ABB RAPID module: Module1.mod

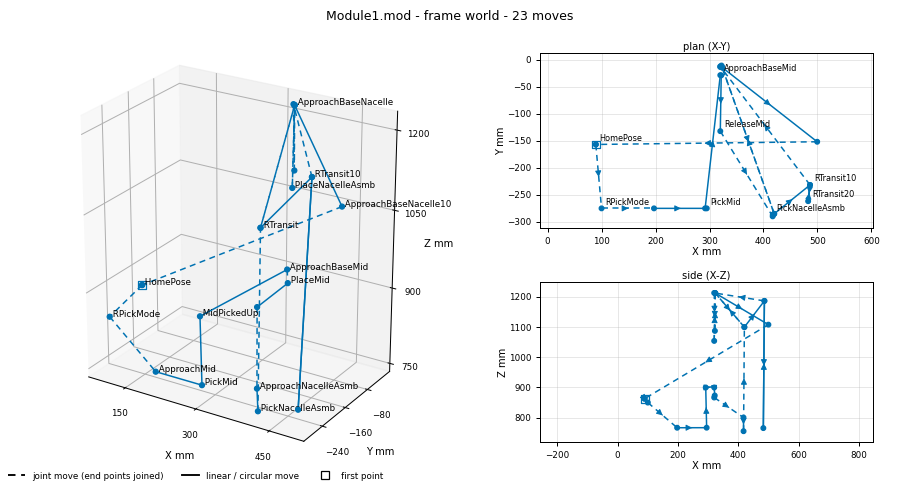
[picture p0: tool path of Module1.mod in frame world, 23 of 23 moves have a stored position in this frame; points joined in program order, loops and branches not executed]
MODULE Module1
    CONST robtarget HomePose:=[[89.387946422,-156.622117956,147.913470217],[0.066010726,-0.842420918,-0.111214912,-0.523068661],[0,0,0,4],[-101.964427132,9E+09,9E+09,9E+09,9E+09,9E+09]];
    CONST robtarget RPickMode:=[[100,-275,135],[0.489762134,0.473830049,0.544432409,0.489092516],[0,0,-1,4],[-101.964427132,9E+09,9E+09,9E+09,9E+09,9E+09]];
    CONST robtarget ApproachMid:=[[-122.697727862,-0.008118871,49.551256125],[0.499992891,0.499992406,0.500008511,0.50000619],[0,0,-1,4],[-101.964431802,9E+09,9E+09,9E+09,9E+09,9E+09]];
    CONST robtarget PickMid:=[[-24.998727784,-0.00024572,49.697076732],[0.499992891,0.499992406,0.500008511,0.50000619],[0,0,-1,4],[-101.964431802,9E+09,9E+09,9E+09,9E+09,9E+09]];
    CONST robtarget MidPickedUp:=[[-27.998642636,0.000176123,182.899085274],[0.499992714,0.499992387,0.500008355,0.500006542],[1,0,-1,4],[-101.964431802,9E+09,9E+09,9E+09,9E+09,9E+09]];
    CONST robtarget ApproachBaseMid:=[[-28.27,0.00,185.00],[0.499997,0.499992,0.500001,0.50001],[1,-1,0,4],[-101.957,9E+09,9E+09,9E+09,9E+09,9E+09]];
    CONST robtarget PlaceMid:=[[-28.61,-1.73,158.37],[0.483819,0.495256,0.51307,0.507346],[1,-1,0,4],[-104.271,9E+09,9E+09,9E+09,9E+09,9E+09]];
    CONST robtarget ReleaseMid:=[[-131.99,0.00,151.74],[0.499992,0.499992,0.500006,0.500009],[1,-1,0,4],[-101.961,9E+09,9E+09,9E+09,9E+09,9E+09]];
    CONST robtarget ApproachNacelleAsmb:=[[15.11,-2.84,84.21],[0.000268004,0.030298,-0.999539,-0.00191911],[1,-2,1,4],[-101.993,9E+09,9E+09,9E+09,9E+09,9E+09]];
    CONST robtarget PickNacelleAsmb:=[[12.03,-2.63,38.86],[4.31501E-05,0.00199455,0.999998,0.00019767],[1,-2,1,4],[-101.924,9E+09,9E+09,9E+09,9E+09,9E+09]];
    CONST robtarget RTransit:=[[-285.112,-99.892,385],[-0.000000669,0.707106579,0.707106983,-0.000001161],[1,-1,0,4],[-101.964431606,9E+09,9E+09,9E+09,9E+09,9E+09]];
    CONST robtarget ApproachBaseNacelle:=[[-13.88,-3.43,497.57],[2.71976E-05,-0.999131,-0.0416698,2.86772E-05],[1,-1,2,4],[-133.038,9E+09,9E+09,9E+09,9E+09,9E+09]];
    CONST robtarget PlaceNacelleAsmb:=[[-13.06,0.09,339.31],[0.00377862,0.999215,0.0389731,0.00594723],[1,-1,2,4],[-132.196,9E+09,9E+09,9E+09,9E+09,9E+09]];
    VAR syncident sync1;
    PERS tasks tasklist1{2}:=[["T_ROB_L"],["T_ROB_R"]];
    VAR syncident sync2;
    VAR syncident sync3;
    CONST robtarget RTransit10:=[[-43.04,66.38,470.53],[2.64793E-06,-0.707288,0.706925,-1.90061E-05],[1,-1,0,4],[-151.87,9E+09,9E+09,9E+09,9E+09,9E+09]];
    CONST robtarget RTransit20:=[[-13.03,62.89,49.13],[5.38536E-05,0.707247,-0.706966,6.14863E-07],[1,-1,0,4],[-144.295,9E+09,9E+09,9E+09,9E+09,9E+09]];
    CONST robtarget ApproachBaseNacelle10:=[[-123.10,79.60,391.87],[0.000794272,0.722511,-0.691359,-0.000251073],[1,-1,1,4],[-150.884,9E+09,9E+09,9E+09,9E+09,9E+09]];
    CONST robtarget ApproachBaseNacelle20:=[[-11.97,0.04,498.20],[0.000211189,0.688434,0.725299,0.000566331],[1,-1,1,4],[-132.988,9E+09,9E+09,9E+09,9E+09,9E+09]];
    CONST robtarget PlaceNacelleAsmb10:=[[-10.40,-2.22,372.47],[0.00176552,-0.688269,-0.725441,-0.00419786],[1,-1,1,4],[-133.194,9E+09,9E+09,9E+09,9E+09,9E+09]];
    VAR syncident sync4;
    PROC Path_10()
        ConfL\Off;
        ConfJ\Off;
        MoveJ HomePose,v500,fine,Servo\WObj:=RightArm;
        MoveJ RPickMode,v100,fine,Servo\WObj:=RightArm;
        g_MoveTo 4;
        MoveJ ApproachMid,v100,fine,Servo\WObj:=MidTower;
        MoveL PickMid,v100,fine,Servo\WObj:=MidTower;
        g_GripIn;
        WaitTime 1;
        MoveL MidPickedUp,v100,fine,Servo\WObj:=MidTower;
        WaitSyncTask\InPos, sync1, tasklist1;
        MoveL ApproachBaseMid,v100,fine,Servo\WObj:=RightTowerBase;
        MoveJ PlaceMid,v100,fine,Servo\WObj:=RightTowerBase;
        g_MoveTo 4;
        WaitTime 1;
        MoveL ReleaseMid,v100,fine,Servo\WObj:=RightTowerBase;
        MoveJ ApproachNacelleAsmb,v100,fine,Servo\WObj:=NacelleAsmb;
        g_MoveTo 15;
        WaitTime 1;
        MoveL PickNacelleAsmb,v100,fine,Servo\WObj:=NacelleAsmb;
        g_GripIn;
        WaitTime 1;
        MoveJ RTransit,v100,fine,Servo\WObj:=RightTowerBase;
        WaitSyncTask\InPos, sync2, tasklist1;
        MoveJ ApproachBaseNacelle,v100,fine,Servo\WObj:=RightTowerBase;
        MoveJ PlaceNacelleAsmb,v100,fine,Servo\WObj:=RightTowerBase;
        g_MoveTo 15;
        WaitTime 1;
        MoveJ ApproachBaseNacelle,v100,fine,Servo\WObj:=RightTowerBase;
        WaitSyncTask\InPos, sync3, tasklist1;
        MoveJ RTransit,v100,fine,Servo\WObj:=RightTowerBase;
        MoveL RTransit10, v100, fine, Servo\WObj:=NacelleAsmb;
        MoveL RTransit20, v100, fine, Servo\WObj:=NacelleAsmb;
        g_GripIn;
        MoveL RTransit10, v100, fine, Servo\WObj:=NacelleAsmb;
        MoveJ ApproachBaseNacelle20, v100, fine, Servo\WObj:=RightTowerBase;
        MoveJ PlaceNacelleAsmb10, v100, fine, Servo\WObj:=RightTowerBase;
        g_MoveTo 15;
        WaitTime 1;
        MoveJ ApproachBaseNacelle,v100,fine,Servo\WObj:=RightTowerBase;
        WaitSyncTask\InPos, sync4, tasklist1;
        MoveL ApproachBaseNacelle10, v100, fine, Servo\WObj:=NacelleAsmb;
        MoveJ HomePose,v500,fine,Servo\WObj:=RightArm;
    ENDPROC
ENDMODULE
